(* PLC project Generated.project, CODESYS CODESYS V3.5 SP19 Patch 1 *)
(* stored: creationDateTime 2026-09-06T13:00:42.534858, modificationDateTime 2026-09-06T13:00:42.534858 *)

(* ═══════════════════════════════════════════════════════════════ 🧲 ST_AcquisitionInterPrg — Bus d'échange inter-PRG produit par PRG_02_Acquisition ─────────────────────────────────────────────────────────────── 🎯 Rôle : Encapsuler les mesures câbles/vitesses, les états joystick qualifiés, les positions M3 et les diagnostics DI publiés par PRG_02_Acquisition vers les consommateurs (PRG_03/04/05/07, FB_TroubleshootingView). 📤 Producteur unique : PRG_02_Acquisition (VAR_OUTPUT Data : ST_AcquisitionInterPrg). 📄 Doc : DOC/AF/AF_Partie-06_Acquisition_Qualification_IO_v2.4.md 🔌 Architecture : Bus de données typé — encapsulation des échanges inter-PRG. ═══════════════════════════════════════════════════════════════ *)
TYPE ST_AcquisitionInterPrg : STRUCT
  DataValid : BOOL;  (* === 🛡️ Drapeau de vie & validité globale des données === 🟢 TRUE = PRG_02 a complété son scan et les données sont fraîches et qualifiées *)
  Joystick : ST_AcquisitionJoystickQualified;  (* === 📦 Structures qualifiées du bus === 🕹️ Données et commandes joystick qualifiées *)
  Network : ST_AcquisitionNetworkDiagnostics;  (* 🔌 Diagnostics réseaux CANopen et EtherCAT *)
  EncoderM1 : ST_AcquisitionEncoderQualified;  (* 🧲 Façade codeur qualifiée M1 (Retenue) *)
  EncoderM2 : ST_AcquisitionEncoderQualified;  (* 🧲 Façade codeur qualifiée M2 (Benne) *)
  MachineHoming : ST_MachineHoming;  (* 🎯 État homing conjoint machine (M1/M2/benne) *)
  InputModules : ST_IOModuleDiag;  (* === 🩺 Diagnostics modules E/S === 🩺 Diagnostic carte des 5 modules E/S (AF06 §3bis) *)
  InputSource : ST_InputSource;  (* === 🧪 Simulation & variateur M3 filtré === 🔀 Flags de bascule de source (réel/simu) par domaine *)
  M3 : ST_M3DriveFeedback;  (* ↔️ Retours variateur M3 filtrés (consommé PRG_05) *)
END_STRUCT;
END_TYPE

(* ═══════════════════════════════════════════════════════════════ 🧲 ST_AcquisitionEncoderQualified — Façade codeur qualifiée ─────────────────────────────────────────────────────────────── 🎯 Rôle : Encapsuler les mesures métriques, statuts de référencement, défauts et signaux hardware produits par FB_Encoder dans PRG_02_Acquisition. 📤 Producteur unique : PRG_02_Acquisition (Data.EncoderM1 / Data.EncoderM2). 📄 Doc : DOC/AF/AF_Partie-06_Acquisition_Qualification_IO_v2.4.md ═══════════════════════════════════════════════════════════════ *)
TYPE ST_AcquisitionEncoderQualified : STRUCT
  Measurement : ST_fbEncoder_Measurement;  (* 📊 Mesure métrique (CablePosM, SpeedMps, etc.) *)
  Ready : BOOL;  (* 🟢 Façade codeur prête *)
  Fault : ST_Fault;  (* ❌ Diagnostic défaut codeur *)
  Homed : BOOL;  (* 🎯 Codeur référencé *)
  HomingSuspect : BOOL;  (* ⚠️ Référencement suspect *)
  EncoderFault : BOOL;  (* ❌ Défaut fiabilité (indisponible ou incohérent) *)
  HomedAndReliable : BOOL;  (* ✅ Référencé ET fiable (sans incohérence) *)
  PresetConfirmationFailed : BOOL;  (* ❌ Échec confirmation preset *)
  HwOut : ST_fbEncoder_HwOut;  (* 📡 Commandes hardware de preset (lecture seule) *)
END_STRUCT;
END_TYPE

(* ═══════════════════════════════════════════════════════════════ 🕹️ ST_AcquisitionJoystickQualified — Données joystick qualifiées ─────────────────────────────────────────────────────────────── 🎯 Rôle : Encapsuler les commandes d'axes, statut homme-mort et diagnostics produits par FB_Joystick dans PRG_02_Acquisition. 📤 Producteur unique : PRG_02_Acquisition (Data.Joystick). 📄 Doc : DOC/AF/AF_Partie-06_Acquisition_Qualification_IO_v2.4.md ═══════════════════════════════════════════════════════════════ *)
TYPE ST_AcquisitionJoystickQualified : STRUCT
  AxisX : ST_fbJoystick_AxisCmd;  (* 📊 Commande et direction qualifiée axe X *)
  AxisY : ST_fbJoystick_AxisCmd;  (* 📊 Commande et direction qualifiée axe Y *)
  DeadmanArmed : BOOL;  (* 🔒 Homme-mort armé et valide *)
  AtNeutralXY : BOOL;  (* 🟢 Les deux axes X et Y sont au neutre *)
  ArmingPermitDenied : BOOL;  (* ⚠️ Tentative d'armement sans permission *)
  Ready : BOOL;  (* 🟢 Façade joystick prête et opérationnelle *)
  Fault : ST_Fault;  (* ❌ Diagnostic défaut joystick *)
  NeutralXAct : INT;  (* 📍 Valeur ADC neutre calibré X *)
  NeutralYAct : INT;  (* 📍 Valeur ADC neutre calibré Y *)
END_STRUCT;
END_TYPE

(* ═══════════════════════════════════════════════════════════════ 🔌 ST_AcquisitionNetworkDiagnostics — Diagnostics réseaux qualifiés ─────────────────────────────────────────────────────────────── 🎯 Rôle : Encapsuler les états opérationnels et diagnostics des bus CANopen et EtherCAT produits par PRG_02_Acquisition. 📤 Producteur unique : PRG_02_Acquisition (Data.Network). 📄 Doc : DOC/AF/AF_Partie-06_Acquisition_Qualification_IO_v2.4.md ═══════════════════════════════════════════════════════════════ *)
TYPE ST_AcquisitionNetworkDiagnostics : STRUCT
  CanOpenMaster : ST_Diag_Device;  (* 🔌 Diagnostic maître CANopen *)
  Joystick : ST_Diag_Device;  (* 🕹️ Diagnostic esclave Joystick MCB560 *)
  EthercatMaster : ST_Diag_Device;  (* 🔌 Diagnostic maître EtherCAT *)
  EncoderM1 : ST_Diag_Device;  (* 🧲 Diagnostic esclave Codeur M1 (COD1) *)
  EncoderM2 : ST_Diag_Device;  (* 🧲 Diagnostic esclave Codeur M2 (COD2) *)
  DriveM3 : ST_Diag_Device;  (* ⚙️ Diagnostic esclave Variateur M3 (AC600) *)
END_STRUCT;
END_TYPE

(* ═══════════════════════════════════════════════════════════════ 🩺 ST_IOModuleDiag — Diagnostic carte des 5 modules E/S physiques ─────────────────────────────────────────────────────────────── 📄 Doc métier : DOC/AF/AF_Partie-06_Acquisition_Qualification_IO_v2.4.md §3bis 🎨 Granularité MODULE (pas canal) : GetDeviceState() est un état de carte, pas un diagnostic par voie. Un module en défaut ne dit pas *quelle* TOR ment, seulement qu'aucune des TOR qu'il porte n'est fiable. 🔗 Producteur : PRG_02_Acquisition (5 appels GetDeviceState()). 🔌 Consommateurs : PRG_04 (SafeStop treuils), PRG_05 (SafeStop M3), PRG_07 (recopie IHM GVL_IHM.Network.InputModules + FB_TroubleshootingView). ═══════════════════════════════════════════════════════════════ *)
TYPE ST_IOModuleDiag : STRUCT
  LocalDigitalIoOk : BOOL;  (* Module Local_Digital_IO OK (DI8/DO8) *)
  Vh0800EndOk : BOOL;  (* Module VH_0800END OK (DI8) *)
  Vh0808EtpOk : BOOL;  (* Module VH_0808ETP OK (DI8/DO8) *)
  Vh0008ErOk : BOOL;  (* Module VH_0008ER OK (DO8 Relais Freins/Kobold) *)
  Vh0008Er1Ok : BOOL;  (* Module VH_0008ER_1 OK (DO8 Relais AU/PowerKeepAlive) *)
  Fault : BOOL;  (* Défaut sur au moins un module E/S *)
END_STRUCT;
END_TYPE

(* ═══════════════════════════════════════════════════════════════ 🔀 ST_InputSource — Flags de bascule de source (réel/simu) par domaine ─────────────────────────────────────────────────────────────── 🎯 Rôle : Regrouper les 4 impulsions 1 cycle signalant qu'une source d'entrée a basculé (réel ↔ simu) pour un domaine donné. 📤 Producteur unique : PRG_02_Acquisition (Data.InputSource). 📥 Consommateur : PRG_07_Supervision (Data.InputSource.* → GVL_IHM). 📄 Doc : DOC/AF/AF_Partie-06_Acquisition_Qualification_IO_v2.4.md 🔌 Architecture : Bus de données typé — encapsulation des échanges inter-PRG. ═══════════════════════════════════════════════════════════════ *)
TYPE ST_InputSource : STRUCT
  WinchInputSourceChanged : BOOL;  (* 🔀 Source Winch a basculé (réel/simu) *)
  TranslationInputSourceChanged : BOOL;  (* 🔀 Source Translation a basculé *)
  OperatorInputSourceChanged : BOOL;  (* 🔀 Source Opérateur a basculé *)
  MachineInputSourceChanged : BOOL;  (* 🔀 Source Machine a basculé *)
END_STRUCT;
END_TYPE

(* ═══════════════════════════════════════════════════════════════ ↔️ ST_M3DriveFeedback — Retours variateur M3 filtrés ─────────────────────────────────────────────────────────────── 🎯 Rôle : Encapsuler les retours variateur M3 (mot d'état + fréquence réelle) conditionnés par PRG_02_Acquisition et consommés par PRG_05_Translation. 📤 Producteur unique : PRG_02_Acquisition (Data.M3). 📥 Consommateur : PRG_05_Translation (Data.M3.StatusWord / Data.M3.ActualFrequencyHz). 📄 Doc : DOC/AF/AF_Partie-06_Acquisition_Qualification_IO_v2.4.md 🔌 Architecture : Bus de données typé — encapsulation des échanges inter-PRG. ═══════════════════════════════════════════════════════════════ *)
TYPE ST_M3DriveFeedback : STRUCT
  StatusWord : UINT;  (* 📊 Mot d'état variateur M3 filtré *)
  ActualFrequencyHz : UINT;  (* 📊 Fréquence réelle M3 filtrée *)
END_STRUCT;
END_TYPE

(* ======================================================================= 🧭 ST_MachineHoming — Etat publie du homing conjoint machine (M1/M2/benne) ─────────────────────────────────────────────────────────────── 🎯 Rôle : Regroupe les 8 sorties homing a plat de PRG_02_Acquisition en un bus struct unique, publie sur le bus inter-PRG. 🔒 Sécurité : Homed = qualification conjointe reference machine (gate SEMI_AUTO). HomingLoss = perte reference en mouvement : arret controle SafeStop. 📄 Doc métier : DOC/AF/AF_Partie-09_Fonction_Encoder_v2.4.md (F09.08) ======================================================================= *)
TYPE ST_MachineHoming : STRUCT
  Homed : BOOL;  (* Qualification conjointe reference machine *)
  SetPosBucketOpen : BOOL;  (* Valider position actuelle = reference benne ouverte *)
  SetPosBucketClose : BOOL;  (* Valider position actuelle = reference benne fermee *)
  Active : BOOL;  (* Homing conjoint en cours *)
  HomingLoss : BOOL;  (* Perte reference en mouvement : arret controle SafeStop *)
  Step : INT;  (* Etape guidee reference (echelle de priorite E_MachineHomingStep) *)
  Instruction : STRING(120);  (* Consigne IHM reference *)
  Failed : BOOL;  (* Transaction reference abandonnee *)
  SeqStep : INT;  (* Step GRAFCET courant (E_MachineHomingTxState HX0..HXF) *)
  M3Locked : BOOL;  (* Translation M3 interdite pendant le cycle de homing machine *)
  CmdWinchM1 : ST_ProgramWinchRequest;  (* Ordre treuil M1 couple palier 1 (HX2 montee / HX3 descente) *)
  CmdWinchM2 : ST_ProgramWinchRequest;  (* Ordre treuil M2 couple palier 1 (HX2 montee / HX3 descente) *)
  CmdBucketOpen : BOOL;  (* Ordre ouverture benne palier 1 sans FDC soft *)
  CmdBucketClose : BOOL;  (* Ordre fermeture benne palier 1 sans FDC soft (HX1) *)
  CmdWinchSelect : INT;  (* Override selecteur treuil cycle homing (-1=neutre, 0=couple, 2=benne) *)
  AllowAscent : BOOL;  (* Autorisation montee par etape GRAFCET homing *)
  AllowDescend : BOOL;  (* Autorisation descente par etape GRAFCET homing *)
  SoftLimitsOff : BOOL;  (* Inhibition limites soft position (HX1..HX3 uniquement, hors capteur TOP) *)
  BucketRefInvalidate : BOOL;  (* Revoque reference benne sur abandon cycle avant HX4 *)
  ProvisionalActive : BOOL;  (* TRUE tant que le zero 0m HX1 est provisoire avant HX4 8.5m *)
  TopContactLatched : BOOL;  (* Contact TOP touche pendant cycle homing : degagement requis *)
  TopContactCount : UINT;  (* Nombre de contacts capteur TOP pendant cycle homing (purge Reset) *)
  ActionText : STRING(120);  (* Consigne d action directe du GRAFCET pour bandeau operateur *)
END_STRUCT;
END_TYPE

(* ======================================================================= 🧩 ST_Fault — Brique socle défaut (2 vues : live + latchée) ─────────────────────────────────────────────────────────────── 🎯 Rôle : porter l'état défaut d'un composant, applicable dans TOUS les cas (acquittable ou non), sans brique warning séparée. • Vue LIVE (Error / ErrorId) : suit la cause, retombe seule à 0. • Vue LATCHÉE (Latched / LatchedId): mémorisée au défaut, reste jusqu'au front Reset. Le choix acquittable / non-acquittable se fait PAR CAUSE (ST_FaultCause.Latching), jamais par bloc. 🔒 Sécurité : interlock TOUJOURS sur la cause brute (Error / ErrorId), jamais sur l'acquittement. Reset TOUJOURS effectif, jamais conditionné (std §9). 🧬 Composition : brique de base réutilisable — sortie de FB, struct métier, GVL. Texte IHM NON stocké ici : dérivé côté IHM depuis LatchedId / ErrorId. 📄 Doc : DOC/STDS/CODE_QUALITY_STANDARDS.md §2quinquies / §9 ======================================================================= *)
TYPE ST_Fault : STRUCT
  Error : BOOL;  (* <-- [DIAG] vue LIVE : au moins une cause présente maintenant *)
  ErrorId : WORD;  (* <-- [DIAG] bitfield des causes présentes maintenant (0 si aucune) *)
  Latched : BOOL;  (* <-- [DIAG] vue LATCHÉE : défaut non acquitté, reste jusqu'au front Reset *)
  LatchedId : WORD;  (* <-- [DIAG] ErrorId figé à l'apparition du défaut, effacé au Reset *)
END_STRUCT;
END_TYPE

(* ======================================================================= 🔌 ST_fbEncoder_HwOut — Ordres preset de sortie codeur (HwOut) ─────────────────────────────────────────────────────────────── 🎯 Rôle : Regrouper les SEULES sorties/ordres preset d'un codeur absolu EtherCAT produits par FB_Encoder vers le PDO Rx (bus sortie). 🔒 Ownership : FB_Encoder produit ce bus ; PRG_02_Acquisition le relaie vers le device. 📄 Doc métier : DOC/AF/AF_Partie-09_Fonction_Encoder_v2.4.md ======================================================================= *)
TYPE ST_fbEncoder_HwOut : STRUCT
  PresetTriggerCmd : WORD;  (* === SORTIES BUS ETHERCAT (ordres preset vers PDO Rx) === <-- [ACT] Declenchement preset vers PDO Rx *)
  CodeSeqTriggerCmd : WORD;  (* <-- [ACT] Sequence code vers PDO Rx, maintenue a 0 *)
  PresetValueOut : UDINT;  (* <-- [ACT] Valeur brute envoyee au preset *)
END_STRUCT;
END_TYPE

(* ======================================================================= 📊 ST_fbEncoder_Measurement — Mesures codeur conditionnées (1 sous-DUT par treuil) ─────────────────────────────────────────────────────────────── 🎯 Rôle : Regroupement des mesures et faits de la chaîne codeur d'un treuil (Abs → Scale → Safety → Speed) 🔌 Interface : Interface de mesure normalisée pour PRG_02_Acquisition 📄 Doc métier : DOC/AF/AF_Partie-06_Acquisition_Qualification_IO_v2.4.md ======================================================================= *)
TYPE ST_fbEncoder_Measurement : STRUCT
  RawPos : UDINT;  (* === DONNEES BRUTES & STATUT BUS === Position brute codeur (gelee si EncoderAvailable=FALSE) *)
  EncoderAvailable : BOOL;  (* TRUE = bus/esclave EtherCAT operationnel et disponible *)
  CablePosM : REAL;  (* === MESURES DE POSITION CABLE === Position cable (m, signee, + enroule) *)
  CablePosMSafe : REAL;  (* Position cable instantanee validee par EncoderIncoherent (m) *)
  EncoderIncoherent : BOOL;  (* TRUE = incoherence redemarrage ou hors bornes *)
  Speed_Mps : REAL;  (* === MESURES DE VITESSE CABLE === Vitesse absolue câble (m/s) *)
  SignedSpeed_Mps : REAL;  (* Vitesse signee câble (m/s, + montee, - descente) *)
  SpeedValid : BOOL;  (* TRUE si mesure valide et codeur operationnel *)
  HomingFault : ST_Fault;  (* === STATUTS DES SOUS-FB & REFERENCE === Défaut FB_Encoder_Homing (état du référencement) *)
  HomingLifecycle : ST_Lifecycle;  (* Cycle FB_Encoder_Homing (Busy/Done) *)
  AbsFault : ST_Fault;  (* Défaut FB_Encoder_Abs (état acquisition bus) *)
  HomingRefRaw : UDINT;  (* Reference brute du dernier homing reussi (re-expose) *)
END_STRUCT;
END_TYPE

(* ======================================================================= 🕹️ ST_fbJoystick_AxisCmd — Consigne d'axe normalisée (sortie FB_Joystick) ─────────────────────────────────────────────────────────────── 🎯 Rôle : Structure de consigne d'axe produite par FB_Joystick. 📤 Champs : Enable, StartStop, SpeedTgt (%) + StepTgt (palier 1..5) + direction en bits (DirectionPositive/Negative, AtNeutral). SpeedTgt reste pour l'IHM, StepTgt pour la logique. 📄 Doc métier : DOC/AF/AF_Partie-08_Fonction_Joystick_v2.5.md ======================================================================= *)
TYPE ST_fbJoystick_AxisCmd : STRUCT
  Enable : BOOL;  (* === CONSIGNES DE PILOTAGE AXE === --> [CMD] Autorisation globale pipeline (FALSE=neutralisation, sorties coupees) *)
  StartStop : BOOL;  (* --> [CMD] Validation de mouvement (TRUE=acceleration, FALSE=deceleration/arret) *)
  SpeedTgt : REAL;  (* --> [CMD] Vitesse cible non signee (0...100 %, signe/sens donné par Direction) - IHM *)
  StepTgt : INT;  (* --> [CMD] Palier de vitesse (1..5, 0=arret) - logique/limitations (derive de SpeedTgt) *)
  DirectionNegative : BOOL;  (* --> [CMD] Direction joystick ou intension de gestuelle *)
  DirectionPositive : BOOL;  (* --> [CMD] Direction joystick ou intension de gestuelle *)
  AtNeutral : BOOL;  (* --> [CMD] TRUE si axes en zone morte (position centrale) *)
  Direction : INT;  (* === MONITORING IHM (derive des bits ci-dessus, jamais lu en interlock) === <-- [STAT] Sens -1=Rev / 0=Neutre / +1=Fwd (anim IHM fleche ; lu aussi logique treuils PRG_04) *)
  Deflection : INT;  (* <-- [STAT] Deflexion signee -100..+100 % (anim IHM jauge/barre) *)
END_STRUCT;
END_TYPE

(* ======================================================================= 📊 ST_Diag_Device — Structure diagnostic d'un esclave ou bus ─────────────────────────────────────────────────────────────── 🎯 Rôle : Structure de donnees d'état, diagnostic et alarme d'un equipement réseau 📄 Doc métier : DOC/AF/AF_Partie-12_Fonction_Diagnostic_v1.4.md ======================================================================= *)
TYPE ST_Diag_Device : STRUCT
  Online : BOOL;  (* Esclave visible sur le bus *)
  Operational : BOOL;  (* Esclave en mode OP (opérationnel) *)
  Error : BOOL;  (* Signal de défaut actif pour cet esclave *)
  ErrorId : WORD;  (* Code défaut détaillé *)
  State : E_Diag_State;  (* Phase courante du cycle de diagnostic *)
  StateAtError : E_Diag_State;  (* Instantané de la phase lors de l'anomalie *)
END_STRUCT;
END_TYPE

(* ======================================================================= 🔌 ST_ProgramWinchRequest — Demande de mouvement treuil par le programme ─────────────────────────────────────────────────────────────── 🎯 Rôle : Regroupe les demandes logiques de treuil formulées par le séquenceur 📄 Référentiel : DOC/WFLOW/CONTRACTS/INTERPRG_CONTRACT_PRG03_MODES_CYCLE_v1.0.md ======================================================================= *)
TYPE ST_ProgramWinchRequest : STRUCT
  RunRequest : BOOL;  (* Ordre marche demandé par le programme *)
  ReqAscent : BOOL;  (* Demande montée *)
  ReqDescend : BOOL;  (* Demande descente *)
  StepTgt : INT;  (* Palier de vitesse cible demandé (1 à 5, 0 = arrêt) *)
END_STRUCT;
END_TYPE

(* ======================================================================= 🧩 ST_Lifecycle — Brique socle cycle d'exécution ─────────────────────────────────────────────────────────────── 🎯 Rôle : porter l'avancement d'une action à cycle (organe, séquenceur). Optionnelle : un FB purement synchrone (conditionneur, filtre, joystick) ne la porte pas. 🧬 Composition : brique de base réutilisable, composée avec ST_Fault. 📄 Doc : DOC/STDS/CODE_QUALITY_STANDARDS.md §2quinquies ======================================================================= *)
TYPE ST_Lifecycle : STRUCT
  Busy : BOOL;  (* <-- [STAT] 1 = action en cours *)
  Done : BOOL;  (* <-- [STAT] 1 = action terminée avec succès *)
END_STRUCT;
END_TYPE

(* values of E_Diag_State: DISABLED: Désactivé (surveillance non active); READY: Opérationnel réel, pas de défaut; INIT: Initialisation / Recherche de réseau; MONITORING: Surveillance active (états transitoires); ERROR: Anomalie de communication; SIMULATED: Bypass simulation ou bypass réseau IHM — pas le bus réel *)

{attribute 'qualified_only'}
{attribute 'strict'}
TYPE E_Diag_State : (DISABLED := 0, READY := 1, INIT := 2, MONITORING := 3, ERROR := 4, SIMULATED := 5);
END_TYPE
